FUNCTION_BLOCK RingTokenControlUnit (* Composite Function Block Type *)
  (* Standard: 61499-2 *)
  (* Version 0.2, 2003-12-05, JHC, Rockwell Automation, Renamed from NEWCOMPFB. *)
  (* Version 0.1, 2002-01-08, JHC, Rockwell Automation, Added DLY FB as example. *)
  (* Version 0.0, 2000-05-27, JHC, Rockwell Automation *)
  (* Compiler header: package fb.rt.cs725; *)
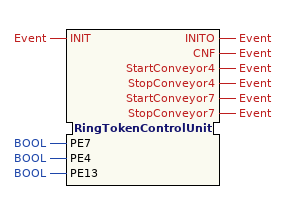
  EVENT_INPUT
    INIT; (* Initialization Request *)
  END_EVENT
  EVENT_OUTPUT
    INITO; (* Initialization Confirm *)
    CNF; (* Execution Confirmation *)
    StartConveyor4;
    StopConveyor4;
    StartConveyor7;
    StopConveyor7;
  END_EVENT
  VAR_INPUT
    PE7 : BOOL;
    PE4 : BOOL;
    PE13 : BOOL;
  END_VAR
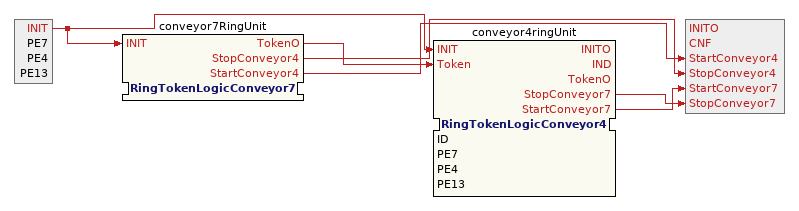
  FBS
    conveyor7RingUnit : RingTokenLogicConveyor7;
    conveyor4ringUnit : RingTokenLogicConveyor4;
  END_FBS
  EVENT_CONNECTIONS
    INIT TO conveyor7RingUnit.INIT;
    INIT TO conveyor4ringUnit.INIT;
    conveyor7RingUnit.TokenO TO conveyor4ringUnit.Token;
    conveyor7RingUnit.StopConveyor4 TO StopConveyor4;
    conveyor7RingUnit.StartConveyor4 TO StartConveyor4;
    conveyor4ringUnit.StopConveyor7 TO StopConveyor7;
    conveyor4ringUnit.StartConveyor7 TO StartConveyor7;
  END_CONNECTIONS
END_FUNCTION_BLOCK
